FUNCTION_BLOCK Pass
  (* Standard: 61499-2 *)
  (* Version 0.1, 2017-00-01, hpea485, UOA *)
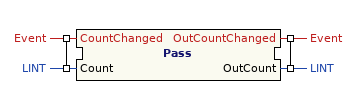
  EVENT_INPUT
    CountChanged WITH Count;
  END_EVENT
  EVENT_OUTPUT
    OutCountChanged WITH OutCount;
  END_EVENT
  VAR_INPUT
    Count : LINT;
  END_VAR
  VAR_OUTPUT
    OutCount : LINT;
  END_VAR
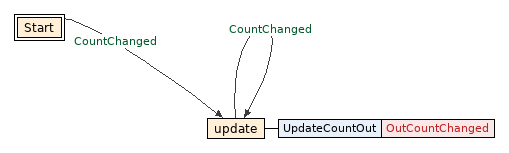
  EC_STATES
    Start;
    update : UpdateCountOut -> OutCountChanged;
  END_STATES
  EC_TRANSITIONS
    Start TO update := CountChanged;
    update TO update := CountChanged;
  END_TRANSITIONS
  ALGORITHM UpdateCountOut IN C:
me->OutCount = me->Count;
  END_ALGORITHM
END_FUNCTION_BLOCK
